Fanuc TP program (LS listing): DOOR_ERR.LS

/PROG  DOOR_ERR
/ATTR
OWNER		= MNEDITOR;
COMMENT		= "";
PROG_SIZE	= 190;
CREATE		= DATE 25-05-27  TIME 12:37:34;
MODIFIED	= DATE 25-07-09  TIME 17:44:34;
FILE_NAME	= T1_RIM_L;
VERSION		= 0;
LINE_COUNT	= 1;
MEMORY_SIZE	= 558;
PROTECT		= READ_WRITE;
TCD:  STACK_SIZE	= 0,
      TASK_PRIORITY	= 50,
      TIME_SLICE	= 0,
      BUSY_LAMP_OFF	= 0,
      ABORT_REQUEST	= 0,
      PAUSE_REQUEST	= 0;
DEFAULT_GROUP	= *,*,*,*,*;
CONTROL_CODE	= 00000000 00000000;
/APPL
/MN
   1:  UALM[2] ;
/POS
/END
